//==================================================================================================
//							Beckhoff Automation Poland
//									23.05.2018
//	Blok funkcyjny kontroli luzownika w silniku podpietym do AX5000. Przewaga ForceLock
//	Datatype:		ENUM (INT16)
//	Enum Value:		0 (0x00): 	Release_force
//					1 (0x01): 	Force_lock
//					2 (0x02): 	Force_unlock
//
// 	v1.1	|| TC v 3.1.4022.16	|| - optymalizacja kodu
//  v1.0	|| TC v 3.1.4022.16	|| - pierwsza wersja
//==================================================================================================
FUNCTION_BLOCK FB_HoldingBrakeCtrlAX5000
VAR_INPUT
	bForceLock 						: BOOL;								// 
	bForceUnlock					: BOOL;								// 
END_VAR
VAR_OUTPUT
	bBusy							: BOOL;
	bError							: BOOL; 							// General error: parameter or CoE read.
																		// If bError = TRUE and bInitialized = FALSE - error during read motor data.
																		// If bError = TRUE and bInitialized = TRUE and (iAdsErrId <> 0 or iCANopenErrId <> 0) then I2T read error
																		// If bError = TRUE and bInitialized = TRUE and iAdsErrId = 0 and iCANopenErrId = 0 then parameter error: rTorqueLimit outside permitted range rTorqueLimitLow..rTorqueLimitHigh or Empty stDriveRef
	iAdsErrId						: UINT;								// Forwarded output FB_SoEWrite
	iSecErrId						: UINT;								// Forwarded output FB_SoEWrite
END_VAR
VAR_IN_OUT
	Axis							: AXIS_REF;
END_VAR
VAR
	bExecute						: BOOL;
	iMotorBrakeForce				: INT;								// 0 - Release_force, 1 - Force_lock, 2 - Force_unlock
	fbSoEWrite						: FB_SoEWrite;
	rtForceLock						: R_TRIG;
	rtForceUnlock					: R_TRIG;
	ftForceLock						: F_TRIG;
	ftForceUnlock					: F_TRIG;
END_VAR

{region "Call triggers"}
//======================= Call triggers =========================
rtForceLock(CLK:= bForceLock);
ftForceLock(CLK:= bForceLock);
rtForceUnlock(CLK:= bForceUnlock);
ftForceUnlock(CLK:= bForceUnlock);
bExecute								:= rtForceLock.Q OR ftForceLock.Q OR rtForceUnlock.Q OR ftForceUnlock.Q;
//===============================================================
{endregion}
{region "Main code"}
//========================= Main code ===========================
IF bExecute THEN
	iMotorBrakeForce 						:= 0;										// Clear value
	iMotorBrakeForce.1 						:= bForceUnlock;							// Set force unlock bit
	iMotorBrakeForce 						:= SEL(bForceLock, iMotorBrakeForce, 1);	// Set force lock bit, it has higher priority than unlock
END_IF
	 
fbSoEWrite(
	NetId			:= '' , 
	Idn				:= P_0_IDN + 96 , 
	Element			:= 16#40 , 
	pSrcBuf			:= ADR(iMotorBrakeForce), 
	BufLen			:= SIZEOF(iMotorBrakeForce) , 
	Execute			:= bExecute , 
	Timeout			:= T#2S, 
	Axis			:= Axis , 
	Busy			=> bBusy , 
	Error			=> bError, 
	AdsErrId		=> iAdsErrId, 
	SercosErrId		=> iSecErrId );
//===============================================================
{endregion}

END_FUNCTION_BLOCK

(* stored: Version 1.1.0.1, ProductVersion 3.1.4022.12
   POU FB_HoldingBrakeCtrlAX5000: Id {c1953c0a-f8e1-44b4-8946-27e90a6eeff4}, SpecialFunc None *)
